Fanuc KAREL source: ka00011.KL

PROGRAM KA00011
%STACKSIZE=65535
%PRIORITY=65535
%NOLOCKGROUP
VAR
SRC : INTEGER
-- UNRESOLVED DECLARATIONS (source type spelling not recovered)
-- DST : ARRAY[2] OF TYPE_0x0018 (type_u16=0x2018)
BEGIN
SRC=2
DST[1]=SRC
END KA00011
